(* CODESYS project Avangard(contr5).project
   Title: Avangard(contr1)
   Version: 0.0.0.0
   Author: Administrator

Project tree, tasks and I/O mapping:
  MyController : TM241CE40T/U, Schneider Electric, order no. TM241CE40T/U, version 4.0.6.18
    application Application
      task MAST (cyclic, interval 20 ms, priority 15, watchdog 100 ms x 1) calls MainPrgY, MainLD, MainPrgX
      global variables GVL
    DI : Digital Inputs, Schneider Electric, version 4.0.6.18
        input  idwDI_IDW0 : DWORD  // IDW0
        input  Application.X05_0 : BOOL  // IDW0.I0
        input  Application.X05_1 : BOOL  // IDW0.I1
        input  Application.X05_2 : BOOL  // IDW0.I2
        input  Application.X05_3 : BOOL  // IDW0.I3
        input  Application.X05_4 : BOOL  // IDW0.I4
        input  Application.X05_5 : BOOL  // IDW0.I5
        input  Application.X05_6 : BOOL  // IDW0.I6
        input  Application.X05_7 : BOOL  // IDW0.I7
        input  Application.X05_8 : BOOL  // IDW0.I8
        input  Application.X05_9 : BOOL  // IDW0.I9
        input  Application.X05_10 : BOOL  // IDW0.I10
        input  Application.X05_11 : BOOL  // IDW0.I11
        input  Application.X05_12 : BOOL  // IDW0.I12
        input  Application.X05_13 : BOOL  // IDW0.I13
        input  Application.X05_14 : BOOL  // IDW0.I14
        input  Application.X05_15 : BOOL  // IDW0.I15
        input  Application.X05_16 : BOOL  // IDW0.I16
        input  Application.X05_17 : BOOL  // IDW0.I17
        input  Application.X05_18 : BOOL  // IDW0.I18
        input  Application.X05_19 : BOOL  // IDW0.I19
        input  Application.X05_20 : BOOL  // IDW0.I20
        input  Application.X05_21 : BOOL  // IDW0.I21
        input  Application.X05_22 : BOOL  // IDW0.I22
        input  Application.X05_23 : BOOL  // IDW0.I23
        input  ibDI_IB1 : BYTE  // IB1
    DQ : Digital Outputs, Schneider Electric, version 4.0.6.18
        output Application.Y05_0 : BOOL  // QW0.Q0
        output Application.Y05_1 : BOOL  // QW0.Q1
        output Application.Y05_2 : BOOL  // QW0.Q2
        output Application.Y05_3 : BOOL  // QW0.Q3
        output Application.Y05_4 : BOOL  // QW0.Q4
        output Application.Y05_5 : BOOL  // QW0.Q5
        output Application.Y05_6 : BOOL  // QW0.Q6
        output Application.Y05_7 : BOOL  // QW0.Q7
        output Application.Y05_8 : BOOL  // QW0.Q8
        output Application.Y05_9 : BOOL  // QW0.Q9
        output Application.Y05_10 : BOOL  // QW0.Q10
        output Application.Y05_11 : BOOL  // QW0.Q11
        output Application.Y05_12 : BOOL  // QW0.Q12
        output Application.Y05_13 : BOOL  // QW0.Q13
        output Application.Y05_14 : BOOL  // QW0.Q14
        output Application.Y05_15 : BOOL  // QW0.Q15
        output qbDQ_QB1 : BYTE  // QB1
        unmapped channels: QW0
    Counters : Counters, Schneider Electric, version 4.0.6.18
    Pulse_Generators : Pulse Generators, Schneider Electric, version 4.0.6.18
    Cartridge_1 : Cartridge, Schneider Electric, version 4.0.6.18
    Cartridge_2 : Cartridge, Schneider Electric, version 4.0.6.18
    IO_Bus : IO bus - TM3, Schneider Electric, version 4.0.6.18
      Module_1 : TM3DI32K, Schneider Electric, order no. TM3DI32K, version 1.0.1.3
          input  idwModule_1_ID0 : DWORD  // ID0
          input  Application.X51_0 : BOOL  // ID0.I0
          input  Application.X51_1 : BOOL  // ID0.I1
          input  Application.X51_2 : BOOL  // ID0.I2
          input  Application.X51_3 : BOOL  // ID0.I3
          input  Application.X51_4 : BOOL  // ID0.I4
          input  Application.X51_5 : BOOL  // ID0.I5
          input  Application.X51_6 : BOOL  // ID0.I6
          input  Application.X51_7 : BOOL  // ID0.I7
          input  Application.X51_8 : BOOL  // ID0.I8
          input  Application.X51_9 : BOOL  // ID0.I9
          input  Application.X51_10 : BOOL  // ID0.I10
          input  Application.X51_11 : BOOL  // ID0.I11
          input  Application.X51_12 : BOOL  // ID0.I12
          input  Application.X51_13 : BOOL  // ID0.I13
          input  Application.X51_14 : BOOL  // ID0.I14
          input  Application.X51_15 : BOOL  // ID0.I15
          input  Application.X51_16 : BOOL  // ID0.I16
          input  Application.X51_17 : BOOL  // ID0.I17
          input  Application.X51_18 : BOOL  // ID0.I18
          input  Application.X51_19 : BOOL  // ID0.I19
          input  Application.X51_20 : BOOL  // ID0.I20
          input  Application.X51_21 : BOOL  // ID0.I21
          input  Application.X51_22 : BOOL  // ID0.I22
          input  Application.X51_23 : BOOL  // ID0.I23
          input  Application.X51_24 : BOOL  // ID0.I24
          input  Application.X51_25 : BOOL  // ID0.I25
          input  Application.X51_26 : BOOL  // ID0.I26
          input  Application.X51_27 : BOOL  // ID0.I27
          input  Application.X51_28 : BOOL  // ID0.I28
          input  Application.X51_29 : BOOL  // ID0.I29
          input  Application.X51_30 : BOOL  // ID0.I30
          input  Application.X51_31 : BOOL  // ID0.I31
      Module_2 : TM3DI32K, Schneider Electric, order no. TM3DI32K, version 1.0.1.3
          input  Application.X52_0 : BOOL  // ID0.I0
          input  Application.X52_1 : BOOL  // ID0.I1
          input  Application.X52_2 : BOOL  // ID0.I2
          input  Application.X52_3 : BOOL  // ID0.I3
          input  Application.X52_4 : BOOL  // ID0.I4
          input  Application.X52_5 : BOOL  // ID0.I5
          input  Application.X52_6 : BOOL  // ID0.I6
          input  Application.X52_7 : BOOL  // ID0.I7
          input  Application.X52_8 : BOOL  // ID0.I8
          input  Application.X52_9 : BOOL  // ID0.I9
          input  Application.X52_10 : BOOL  // ID0.I10
          input  Application.X52_11 : BOOL  // ID0.I11
          input  Application.X52_12 : BOOL  // ID0.I12
          input  Application.X52_13 : BOOL  // ID0.I13
          input  Application.X52_14 : BOOL  // ID0.I14
          input  Application.X52_15 : BOOL  // ID0.I15
          input  Application.X52_16 : BOOL  // ID0.I16
          input  Application.X52_17 : BOOL  // ID0.I17
          input  Application.X52_18 : BOOL  // ID0.I18
          input  Application.X52_19 : BOOL  // ID0.I19
          input  Application.X52_20 : BOOL  // ID0.I20
          input  Application.X52_21 : BOOL  // ID0.I21
          input  Application.X52_22 : BOOL  // ID0.I22
          input  Application.X52_23 : BOOL  // ID0.I23
          input  Application.X52_24 : BOOL  // ID0.I24
          input  Application.X52_25 : BOOL  // ID0.I25
          input  Application.X52_26 : BOOL  // ID0.I26
          input  Application.X52_27 : BOOL  // ID0.I27
          input  Application.X52_28 : BOOL  // ID0.I28
          input  Application.X52_29 : BOOL  // ID0.I29
          input  Application.X52_30 : BOOL  // ID0.I30
          input  Application.X52_31 : BOOL  // ID0.I31
          unmapped channels: ID0
      Module_7 : TM3TI4/G, Schneider Electric, order no. TM3TI4/G, version 1.0.1.5
          input  Application.XXa7_0 : INT  // IW0
          input  Application.XXa7_1 : INT  // IW1
          input  Application.XXa7_2 : INT  // IW2
          input  Application.XXa7_3 : INT  // IW3
          input  ibModule_9_IBStatusIW0 : BYTE  // IBStatusIW0
          input  ibModule_9_IBStatusIW1 : BYTE  // IBStatusIW1
          input  ibModule_9_IBStatusIW2 : BYTE  // IBStatusIW2
          input  ibModule_9_IBStatusIW3 : BYTE  // IBStatusIW3
      Module_4 : TM3DI32K, Schneider Electric, order no. TM3DI32K, version 1.0.1.3
          input  Application.X54_0 : BOOL  // ID0.I0
          input  Application.X54_1 : BOOL  // ID0.I1
          input  Application.X54_2 : BOOL  // ID0.I2
          input  Application.X54_3 : BOOL  // ID0.I3
          input  Application.X54_4 : BOOL  // ID0.I4
          input  Application.X54_5 : BOOL  // ID0.I5
          input  Application.X54_6 : BOOL  // ID0.I6
          input  Application.X54_7 : BOOL  // ID0.I7
          input  Application.X54_8 : BOOL  // ID0.I8
          input  Application.X54_9 : BOOL  // ID0.I9
          input  Application.X54_10 : BOOL  // ID0.I10
          input  Application.X54_11 : BOOL  // ID0.I11
          input  Application.X54_12 : BOOL  // ID0.I12
          input  Application.X54_13 : BOOL  // ID0.I13
          input  Application.X54_14 : BOOL  // ID0.I14
          input  Application.X54_15 : BOOL  // ID0.I15
          input  Application.X54_16 : BOOL  // ID0.I16
          input  Application.X54_17 : BOOL  // ID0.I17
          input  Application.X54_18 : BOOL  // ID0.I18
          input  Application.X54_19 : BOOL  // ID0.I19
          input  Application.X54_20 : BOOL  // ID0.I20
          input  Application.X54_21 : BOOL  // ID0.I21
          input  Application.X54_22 : BOOL  // ID0.I22
          input  Application.X54_23 : BOOL  // ID0.I23
          input  Application.X54_24 : BOOL  // ID0.I24
          input  Application.X54_25 : BOOL  // ID0.I25
          input  Application.X54_26 : BOOL  // ID0.I26
          input  Application.X54_27 : BOOL  // ID0.I27
          input  Application.X54_28 : BOOL  // ID0.I28
          input  Application.X54_29 : BOOL  // ID0.I29
          input  Application.X54_30 : BOOL  // ID0.I30
          input  Application.X54_31 : BOOL  // ID0.I31
          unmapped channels: ID0
      Module_3 : TM3DI32K, Schneider Electric, order no. TM3DI32K, version 1.0.1.3
          input  Application.X53_0 : BOOL  // ID0.I0
          input  Application.X53_1 : BOOL  // ID0.I1
          input  Application.X53_2 : BOOL  // ID0.I2
          input  Application.X53_3 : BOOL  // ID0.I3
          input  Application.X53_4 : BOOL  // ID0.I4
          input  Application.X53_5 : BOOL  // ID0.I5
          input  Application.X53_6 : BOOL  // ID0.I6
          input  Application.X53_7 : BOOL  // ID0.I7
          input  Application.X53_8 : BOOL  // ID0.I8
          input  Application.X53_9 : BOOL  // ID0.I9
          input  Application.X53_10 : BOOL  // ID0.I10
          input  Application.X53_11 : BOOL  // ID0.I11
          input  Application.X53_12 : BOOL  // ID0.I12
          input  Application.X53_13 : BOOL  // ID0.I13
          input  Application.X53_14 : BOOL  // ID0.I14
          input  Application.X53_15 : BOOL  // ID0.I15
          input  Application.X53_16 : BOOL  // ID0.I16
          input  Application.X53_17 : BOOL  // ID0.I17
          input  Application.X53_18 : BOOL  // ID0.I18
          input  Application.X53_19 : BOOL  // ID0.I19
          input  Application.X53_20 : BOOL  // ID0.I20
          input  Application.X53_21 : BOOL  // ID0.I21
          input  Application.X53_22 : BOOL  // ID0.I22
          input  Application.X53_23 : BOOL  // ID0.I23
          input  Application.X53_24 : BOOL  // ID0.I24
          input  Application.X53_25 : BOOL  // ID0.I25
          input  Application.X53_26 : BOOL  // ID0.I26
          input  Application.X53_27 : BOOL  // ID0.I27
          input  Application.X53_28 : BOOL  // ID0.I28
          input  Application.X53_29 : BOOL  // ID0.I29
          input  Application.X53_30 : BOOL  // ID0.I30
          input  Application.X53_31 : BOOL  // ID0.I31
          unmapped channels: ID0
      Module_5 : TM3DQ32TK, Schneider Electric, order no. TM3DQ32TK, version 1.0.1.3
          output Application.Y55_0 : BOOL  // QD0.Q0
          output Application.Y55_1 : BOOL  // QD0.Q1
          output Application.Y55_2 : BOOL  // QD0.Q2
          output Application.Y55_3 : BOOL  // QD0.Q3
          output Application.Y55_4 : BOOL  // QD0.Q4
          output Application.Y55_5 : BOOL  // QD0.Q5
          output Application.Y55_6 : BOOL  // QD0.Q6
          output Application.Y55_7 : BOOL  // QD0.Q7
          output Application.Y55_8 : BOOL  // QD0.Q8
          output Application.Y55_9 : BOOL  // QD0.Q9
          output Application.Y55_10 : BOOL  // QD0.Q10
          output Application.Y55_11 : BOOL  // QD0.Q11
          output Application.Y55_12 : BOOL  // QD0.Q12
          output Application.Y55_13 : BOOL  // QD0.Q13
          output Application.Y55_14 : BOOL  // QD0.Q14
          output Application.Y55_15 : BOOL  // QD0.Q15
          output Application.Y55_16 : BOOL  // QD0.Q16
          output Application.Y55_17 : BOOL  // QD0.Q17
          output Application.Y55_18 : BOOL  // QD0.Q18
          output Application.Y55_19 : BOOL  // QD0.Q19
          output Application.Y55_20 : BOOL  // QD0.Q20
          output Application.Y55_21 : BOOL  // QD0.Q21
          output Application.Y55_22 : BOOL  // QD0.Q22
          output Application.Y55_23 : BOOL  // QD0.Q23
          output Application.Y55_24 : BOOL  // QD0.Q24
          output Application.Y55_25 : BOOL  // QD0.Q25
          output Application.Y55_26 : BOOL  // QD0.Q26
          output Application.Y55_27 : BOOL  // QD0.Q27
          output Application.Y55_28 : BOOL  // QD0.Q28
          output Application.Y55_29 : BOOL  // QD0.Q29
          output Application.Y55_30 : BOOL  // QD0.Q30
          output Application.Y55_31 : BOOL  // QD0.Q31
          unmapped channels: QD0
      Module_6 : TM3TI4/G, Schneider Electric, order no. TM3TI4/G, version 1.0.1.5
          input  Application.XXa6_0 : INT  // IW0
          input  Application.XXa6_1 : INT  // IW1
          input  Application.XXa6_2 : INT  // IW2
          input  Application.XXa6_3 : INT  // IW3
          input  ibModule_8_IBStatusIW0 : BYTE  // IBStatusIW0
          input  ibModule_8_IBStatusIW1 : BYTE  // IBStatusIW1
          input  ibModule_8_IBStatusIW2 : BYTE  // IBStatusIW2
          input  ibModule_8_IBStatusIW3 : BYTE  // IBStatusIW3
    COM_Bus : COM bus, Schneider Electric, version 4.0.6.18
    Ethernet_1 : Ethernet Network, Schneider Electric, version 4.0.6.18
        settings: IPAddress = [192, 168, 1, 205]; SubnetMask = [255, 255, 255, 0]; GatewayAddress = [192, 168, 1, 1]; DeviceName = 'TM241CE40T_5'; WebServer = FALSE; FTP Server = FALSE; SoMachine Protocol = TRUE; Modbus Server = TRUE; NetManage Protocol = TRUE; SNMP protocol = FALSE; Enable Routing = FALSE; WebVisu protocol = FALSE; DHCP Server Active = FALSE
    Serial_Line_1 : Serial line, Schneider Electric, version 4.0.6.18
      SoMachine_Network_Manager : SoMachine-Network Manager, Schneider Electric, version 4.0.0.2
    Serial_Line_2 : Serial line, Schneider Electric, version 4.0.6.18
      Modbus_Manager : Modbus Manager, Schneider Electric, version 4.0.0.2
  libraries: Standard, * (System)
  program MainPrgY [ST]
  program MainLD [LD]
  function block DKS [LD]
  program MainPrgX [ST]
*)

// MyController/Application/GVL
VAR_GLOBAL
	XX AT %MW0 : ARRAY[0..9] OF WORD;  //данные с 5го контроллера
	XXa AT %MW10 : ARRAY[0..8] OF INT;  //данные с 5го контроллера
	YY AT %MW18 : ARRAY[0..3] OF WORD;  //данные для 5го контроллера на управление

	DKS_Time : WORD := 3;	//время срабатывания ДКС в сек
	
	Nor10200_DKS : BOOL;
	Nor10400_DKS : BOOL;
	Tr10500_DKS : BOOL;
	Tr10600_DKS : BOOL;
	Tr10700_DKS : BOOL;
	Tr20110_DKS : BOOL;
	Nor20300_DKS : BOOL;
	Nor21200_DKS : BOOL;
	Tr21300_DKS : BOOL;
	Tr30400_DKS : BOOL;
	Nor30500_DKS : BOOL;
	Tr30340_DKS : BOOL;
	Tr30700_DKS : BOOL;
	Nor40100_DKS : BOOL;
	
	
	// Контроллер 1
		//Входа
			X05_0 : BOOL;
			X05_1 : BOOL;
			X05_2 : BOOL;
			X05_3 : BOOL;
			X05_4 : BOOL;
			X05_5 : BOOL;
			X05_6 : BOOL;
			X05_7 : BOOL;
			X05_8 : BOOL;
			X05_9 : BOOL;
			X05_10 : BOOL;
			X05_11 : BOOL;
			X05_12 : BOOL;
			X05_13 : BOOL;
			X05_14 : BOOL;
			X05_15 : BOOL;
			X05_16 : BOOL;
			X05_17 : BOOL;
			X05_18 : BOOL;
			X05_19 : BOOL;
			X05_20 : BOOL;
			X05_21 : BOOL;
			X05_22 : BOOL;
			X05_23 : BOOL;
			X05_24 : BOOL;
			X05_25 : BOOL;
			X05_26 : BOOL;
			X05_27 : BOOL;
			X05_28 : BOOL;
			X05_29 : BOOL;
			X05_30 : BOOL;
			X05_31 : BOOL;
		//Выхода
			Y05_0 : BOOL;
			Y05_1 : BOOL;
			Y05_2 : BOOL;
			Y05_3 : BOOL;
			Y05_4 : BOOL;
			Y05_5 : BOOL;
			Y05_6 : BOOL;
			Y05_7 : BOOL;
			Y05_8 : BOOL;
			Y05_9 : BOOL;
			Y05_10 : BOOL;
			Y05_11 : BOOL;
			Y05_12 : BOOL;
			Y05_13 : BOOL;
			Y05_14 : BOOL;
			Y05_15 : BOOL;
			Y05_16 : BOOL;
			Y05_17 : BOOL;
			Y05_18 : BOOL;
			Y05_19 : BOOL;
			Y05_20 : BOOL;
			Y05_21 : BOOL;
			Y05_22 : BOOL;
			Y05_23 : BOOL;
			Y05_24 : BOOL;
			Y05_25 : BOOL;
			Y05_26 : BOOL;
			Y05_27 : BOOL;
			Y05_28 : BOOL;
			Y05_29 : BOOL;
			Y05_30 : BOOL;
			Y05_31 : BOOL;
			
	// Модуль расширения 1 контроллер 1 
		//Входа
			X51_0 : BOOL;
			X51_1 : BOOL;
			X51_2 : BOOL;
			X51_3 : BOOL;
			X51_4 : BOOL;
			X51_5 : BOOL;
			X51_6 : BOOL;
			X51_7 : BOOL;
			X51_8 : BOOL;
			X51_9 : BOOL;
			X51_10 : BOOL;
			X51_11 : BOOL;
			X51_12 : BOOL;
			X51_13 : BOOL;
			X51_14 : BOOL;
			X51_15 : BOOL;
			X51_16 : BOOL;
			X51_17 : BOOL;
			X51_18 : BOOL;
			X51_19 : BOOL;
			X51_20 : BOOL;
			X51_21 : BOOL;
			X51_22 : BOOL;
			X51_23 : BOOL;
			X51_24 : BOOL;
			X51_25 : BOOL;
			X51_26 : BOOL;
			X51_27 : BOOL;
			X51_28 : BOOL;
			X51_29 : BOOL;
			X51_30 : BOOL;
			X51_31 : BOOL;
		//Выхода
			Y51_0 : BOOL;
			Y51_1 : BOOL;
			Y51_2 : BOOL;
			Y51_3 : BOOL;
			Y51_4 : BOOL;
			Y51_5 : BOOL;
			Y51_6 : BOOL;
			Y51_7 : BOOL;
			Y51_8 : BOOL;
			Y51_9 : BOOL;
			Y51_10 : BOOL;
			Y51_11 : BOOL;
			Y51_12 : BOOL;
			Y51_13 : BOOL;
			Y51_14 : BOOL;
			Y51_15 : BOOL;
			Y51_16 : BOOL;
			Y51_17 : BOOL;
			Y51_18 : BOOL;
			Y51_19 : BOOL;
			Y51_20 : BOOL;
			Y51_21 : BOOL;
			Y51_22 : BOOL;
			Y51_23 : BOOL;
			Y51_24 : BOOL;
			Y51_25 : BOOL;
			Y51_26 : BOOL;
			Y51_27 : BOOL;
			Y51_28 : BOOL;
			Y51_29 : BOOL;
			Y51_30 : BOOL;
			Y51_31 : BOOL;
	
	// Модуль расширения 2 контроллер 1
		//Входа
			X52_0 : BOOL;
			X52_1 : BOOL;
			X52_2 : BOOL;
			X52_3 : BOOL;
			X52_4 : BOOL;
			X52_5 : BOOL;
			X52_6 : BOOL;
			X52_7 : BOOL;
			X52_8 : BOOL;
			X52_9 : BOOL;
			X52_10 : BOOL;
			X52_11 : BOOL;
			X52_12 : BOOL;
			X52_13 : BOOL;
			X52_14 : BOOL;
			X52_15 : BOOL;
			X52_16 : BOOL;
			X52_17 : BOOL;
			X52_18 : BOOL;
			X52_19 : BOOL;
			X52_20 : BOOL;
			X52_21 : BOOL;
			X52_22 : BOOL;
			X52_23 : BOOL;
			X52_24 : BOOL;
			X52_25 : BOOL;
			X52_26 : BOOL;
			X52_27 : BOOL;
			X52_28 : BOOL;
			X52_29 : BOOL;
			X52_30 : BOOL;
			X52_31 : BOOL;
		//Выхода
			Y52_0 : BOOL;
			Y52_1 : BOOL;
			Y52_2 : BOOL;
			Y52_3 : BOOL;
			Y52_4 : BOOL;
			Y52_5 : BOOL;
			Y52_6 : BOOL;
			Y52_7 : BOOL;
			Y52_8 : BOOL;
			Y52_9 : BOOL;
			Y52_10 : BOOL;
			Y52_11 : BOOL;
			Y52_12 : BOOL;
			Y52_13 : BOOL;
			Y52_14 : BOOL;
			Y52_15 : BOOL;
			Y52_16 : BOOL;
			Y52_17 : BOOL;
			Y52_18 : BOOL;
			Y52_19 : BOOL;
			Y52_20 : BOOL;
			Y52_21 : BOOL;
			Y52_22 : BOOL;
			Y52_23 : BOOL;
			Y52_24 : BOOL;
			Y52_25 : BOOL;
			Y52_26 : BOOL;
			Y52_27 : BOOL;
			Y52_28 : BOOL;
			Y52_29 : BOOL;
			Y52_30 : BOOL;
			Y52_31 : BOOL;
			
	// Модуль расширения 3 контроллер 1
		//Входа
			X53_0 : BOOL;
			X53_1 : BOOL;
			X53_2 : BOOL;
			X53_3 : BOOL;
			X53_4 : BOOL;
			X53_5 : BOOL;
			X53_6 : BOOL;
			X53_7 : BOOL;
			X53_8 : BOOL;
			X53_9 : BOOL;
			X53_10 : BOOL;
			X53_11 : BOOL;
			X53_12 : BOOL;
			X53_13 : BOOL;
			X53_14 : BOOL;
			X53_15 : BOOL;
			X53_16 : BOOL;
			X53_17 : BOOL;
			X53_18 : BOOL;
			X53_19 : BOOL;
			X53_20 : BOOL;
			X53_21 : BOOL;
			X53_22 : BOOL;
			X53_23 : BOOL;
			X53_24 : BOOL;
			X53_25 : BOOL;
			X53_26 : BOOL;
			X53_27 : BOOL;
			X53_28 : BOOL;
			X53_29 : BOOL;
			X53_30 : BOOL;
			X53_31 : BOOL;
		//Выхода
			Y53_0 : BOOL;
			Y53_1 : BOOL;
			Y53_2 : BOOL;
			Y53_3 : BOOL;
			Y53_4 : BOOL;
			Y53_5 : BOOL;
			Y53_6 : BOOL;
			Y53_7 : BOOL;
			Y53_8 : BOOL;
			Y53_9 : BOOL;
			Y53_10 : BOOL;
			Y53_11 : BOOL;
			Y53_12 : BOOL;
			Y53_13 : BOOL;
			Y53_14 : BOOL;
			Y53_15 : BOOL;
			Y53_16 : BOOL;
			Y53_17 : BOOL;
			Y53_18 : BOOL;
			Y53_19 : BOOL;
			Y53_20 : BOOL;
			Y53_21 : BOOL;
			Y53_22 : BOOL;
			Y53_23 : BOOL;
			Y53_24 : BOOL;
			Y53_25 : BOOL;
			Y53_26 : BOOL;
			Y53_27 : BOOL;
			Y53_28 : BOOL;
			Y53_29 : BOOL;
			Y53_30 : BOOL;
			Y53_31 : BOOL;			

	// Модуль расширения 4 контроллер 1
		//Входа
			X54_0 : BOOL;
			X54_1 : BOOL;
			X54_2 : BOOL;
			X54_3 : BOOL;
			X54_4 : BOOL;
			X54_5 : BOOL;
			X54_6 : BOOL;
			X54_7 : BOOL;
			X54_8 : BOOL;
			X54_9 : BOOL;
			X54_10 : BOOL;
			X54_11 : BOOL;
			X54_12 : BOOL;
			X54_13 : BOOL;
			X54_14 : BOOL;
			X54_15 : BOOL;
			X54_16 : BOOL;
			X54_17 : BOOL;
			X54_18 : BOOL;
			X54_19 : BOOL;
			X54_20 : BOOL;
			X54_21 : BOOL;
			X54_22 : BOOL;
			X54_23 : BOOL;
			X54_24 : BOOL;
			X54_25 : BOOL;
			X54_26 : BOOL;
			X54_27 : BOOL;
			X54_28 : BOOL;
			X54_29 : BOOL;
			X54_30 : BOOL;
			X54_31 : BOOL;
		//Выхода
			Y54_0 : BOOL;
			Y54_1 : BOOL;
			Y54_2 : BOOL;
			Y54_3 : BOOL;
			Y54_4 : BOOL;
			Y54_5 : BOOL;
			Y54_6 : BOOL;
			Y54_7 : BOOL;
			Y54_8 : BOOL;
			Y54_9 : BOOL;
			Y54_10 : BOOL;
			Y54_11 : BOOL;
			Y54_12 : BOOL;
			Y54_13 : BOOL;
			Y54_14 : BOOL;
			Y54_15 : BOOL;
			Y54_16 : BOOL;
			Y54_17 : BOOL;
			Y54_18 : BOOL;
			Y54_19 : BOOL;
			Y54_20 : BOOL;
			Y54_21 : BOOL;
			Y54_22 : BOOL;
			Y54_23 : BOOL;
			Y54_24 : BOOL;
			Y54_25 : BOOL;
			Y54_26 : BOOL;
			Y54_27 : BOOL;
			Y54_28 : BOOL;
			Y54_29 : BOOL;
			Y54_30 : BOOL;
			Y54_31 : BOOL;
	// Модуль расширения 5 контроллер 1
		//Входа
			X55_0 : BOOL;
			X55_1 : BOOL;
			X55_2 : BOOL;
			X55_3 : BOOL;
			X55_4 : BOOL;
			X55_5 : BOOL;
			X55_6 : BOOL;
			X55_7 : BOOL;
			X55_8 : BOOL;
			X55_9 : BOOL;
			X55_10 : BOOL;
			X55_11 : BOOL;
			X55_12 : BOOL;
			X55_13 : BOOL;
			X55_14 : BOOL;
			X55_15 : BOOL;
			X55_16 : BOOL;
			X55_17 : BOOL;
			X55_18 : BOOL;
			X55_19 : BOOL;
			X55_20 : BOOL;
			X55_21 : BOOL;
			X55_22 : BOOL;
			X55_23 : BOOL;
			X55_24 : BOOL;
			X55_25 : BOOL;
			X55_26 : BOOL;
			X55_27 : BOOL;
			X55_28 : BOOL;
			X55_29 : BOOL;
			X55_30 : BOOL;
			X55_31 : BOOL;
		//Выхода
			Y55_0 : BOOL;
			Y55_1 : BOOL;
			Y55_2 : BOOL;
			Y55_3 : BOOL;
			Y55_4 : BOOL;
			Y55_5 : BOOL;
			Y55_6 : BOOL;
			Y55_7 : BOOL;
			Y55_8 : BOOL;
			Y55_9 : BOOL;
			Y55_10 : BOOL;
			Y55_11 : BOOL;
			Y55_12 : BOOL;
			Y55_13 : BOOL;
			Y55_14 : BOOL;
			Y55_15 : BOOL;
			Y55_16 : BOOL;
			Y55_17 : BOOL;
			Y55_18 : BOOL;
			Y55_19 : BOOL;
			Y55_20 : BOOL;
			Y55_21 : BOOL;
			Y55_22 : BOOL;
			Y55_23 : BOOL;
			Y55_24 : BOOL;
			Y55_25 : BOOL;
			Y55_26 : BOOL;
			Y55_27 : BOOL;
			Y55_28 : BOOL;
			Y55_29 : BOOL;
			Y55_30 : BOOL;
			Y55_31 : BOOL;
	// Модуль расширения 6 контроллер 1
		//Входа
			X56_0 : BOOL;
			X56_1 : BOOL;
			X56_2 : BOOL;
			X56_3 : BOOL;
			X56_4 : BOOL;
			X56_5 : BOOL;
			X56_6 : BOOL;
			X56_7 : BOOL;
			X56_8 : BOOL;
			X56_9 : BOOL;
			X56_10 : BOOL;
			X56_11 : BOOL;
			X56_12 : BOOL;
			X56_13 : BOOL;
			X56_14 : BOOL;
			X56_15 : BOOL;
			X56_16 : BOOL;
			X56_17 : BOOL;
			X56_18 : BOOL;
			X56_19 : BOOL;
			X56_20 : BOOL;
			X56_21 : BOOL;
			X56_22 : BOOL;
			X56_23 : BOOL;
			X56_24 : BOOL;
			X56_25 : BOOL;
			X56_26 : BOOL;
			X56_27 : BOOL;
			X56_28 : BOOL;
			X56_29 : BOOL;
			X56_30 : BOOL;
			X56_31 : BOOL;
		//Выхода
			Y56_0 : BOOL;
			Y56_1 : BOOL;
			Y56_2 : BOOL;
			Y56_3 : BOOL;
			Y56_4 : BOOL;
			Y56_5 : BOOL;
			Y56_6 : BOOL;
			Y56_7 : BOOL;
			Y56_8 : BOOL;
			Y56_9 : BOOL;
			Y56_10 : BOOL;
			Y56_11 : BOOL;
			Y56_12 : BOOL;
			Y56_13 : BOOL;
			Y56_14 : BOOL;
			Y56_15 : BOOL;
			Y56_16 : BOOL;
			Y56_17 : BOOL;
			Y56_18 : BOOL;
			Y56_19 : BOOL;
			Y56_20 : BOOL;
			Y56_21 : BOOL;
			Y56_22 : BOOL;
			Y56_23 : BOOL;
			Y56_24 : BOOL;
			Y56_25 : BOOL;
			Y56_26 : BOOL;
			Y56_27 : BOOL;
			Y56_28 : BOOL;
			Y56_29 : BOOL;
			Y56_30 : BOOL;
			Y56_31 : BOOL;

	// Модуль расширения 7 контроллер 1
		//Входа
			X57_0 : BOOL;
			X57_1 : BOOL;
			X57_2 : BOOL;
			X57_3 : BOOL;
			X57_4 : BOOL;
			X57_5 : BOOL;
			X57_6 : BOOL;
			X57_7 : BOOL;
			X57_8 : BOOL;
			X57_9 : BOOL;
			X57_10 : BOOL;
			X57_11 : BOOL;
			X57_12 : BOOL;
			X57_13 : BOOL;
			X57_14 : BOOL;
			X57_15 : BOOL;
			X57_16 : BOOL;
			X57_17 : BOOL;
			X57_18 : BOOL;
			X57_19 : BOOL;
			X57_20 : BOOL;
			X57_21 : BOOL;
			X57_22 : BOOL;
			X57_23 : BOOL;
			X57_24 : BOOL;
			X57_25 : BOOL;
			X57_26 : BOOL;
			X57_27 : BOOL;
			X57_28 : BOOL;
			X57_29 : BOOL;
			X57_30 : BOOL;
			X57_31 : BOOL;
		//Выхода
			Y57_0 : BOOL;
			Y57_1 : BOOL;
			Y57_2 : BOOL;
			Y57_3 : BOOL;
			Y57_4 : BOOL;
			Y57_5 : BOOL;
			Y57_6 : BOOL;
			Y57_7 : BOOL;
			Y57_8 : BOOL;
			Y57_9 : BOOL;
			Y57_10 : BOOL;
			Y57_11 : BOOL;
			Y57_12 : BOOL;
			Y57_13 : BOOL;
			Y57_14 : BOOL;
			Y57_15 : BOOL;
			Y57_16 : BOOL;
			Y57_17 : BOOL;
			Y57_18 : BOOL;
			Y57_19 : BOOL;
			Y57_20 : BOOL;
			Y57_21 : BOOL;
			Y57_22 : BOOL;
			Y57_23 : BOOL;
			Y57_24 : BOOL;
			Y57_25 : BOOL;
			Y57_26 : BOOL;
			Y57_27 : BOOL;
			Y57_28 : BOOL;
			Y57_29 : BOOL;
			Y57_30 : BOOL;
			Y57_31 : BOOL;
			
	XXa6_0 : INT;
	XXa6_1 : INT;
	XXa6_2 : INT;
	XXa6_3 : INT;
	XXa7_0 : INT;
	XXa7_1 : INT;
	XXa7_2 : INT;
	XXa7_3 : INT;

END_VAR

// MainPrgY
PROGRAM MainPrgY
VAR
END_VAR

	//выходы
		Y05_0 := YY[0].0;		
		Y05_1 := YY[0].1;
		Y05_2 := YY[0].2;
		Y05_3 := YY[0].3;
		Y05_4 := YY[0].4;
		Y05_5 := YY[0].5;
		Y05_6 := YY[0].6;
		Y05_7 := YY[0].7;
		Y05_8 := YY[0].8;
		Y05_9 := YY[0].9;
		Y05_10 := YY[0].10;
		Y05_11 := YY[0].11;
		Y05_12 := YY[0].12;
		Y05_13 := YY[0].13;
		Y05_14 := YY[0].14;
		Y05_15 := YY[0].15;
		Y05_16 := YY[1].0;
		Y05_17 := YY[1].1;
		Y05_18 := YY[1].2;
		Y05_19 := YY[1].3;
		Y05_20 := YY[1].4;
		Y05_21 := YY[1].5;
		Y05_22 := YY[1].6;
		Y05_23 := YY[1].7;
		Y05_24 := YY[1].8;
		Y05_25 := YY[1].9;
		Y05_26 := YY[1].10;
		Y05_27 := YY[1].11;
		Y05_28 := YY[1].12;
		Y05_29 := YY[1].13;
		Y05_30 := YY[1].14;
		Y05_31 := YY[1].15;
		
		Y55_0 := YY[2].0;		
		Y55_1 := YY[2].1;
		Y55_2 := YY[2].2;
		Y55_3 := YY[2].3;
		Y55_4 := YY[2].4;
		Y55_5 := YY[2].5;
		Y55_6 := YY[2].6;
		Y55_7 := YY[2].7;
		Y55_8 := YY[2].8;
		Y55_9 := YY[2].9;
		Y55_10 := YY[2].10;
		Y55_11 := YY[2].11;
		Y55_12 := YY[2].12;
		Y55_13 := YY[2].13;
		Y55_14 := YY[2].14;
		Y55_15 := YY[2].15;
		Y55_16 := YY[3].0;
		Y55_17 := YY[3].1;
		Y55_18 := YY[3].2;
		Y55_19 := YY[3].3;
		Y55_20 := YY[3].4;
		Y55_21 := YY[3].5;
		Y55_22 := YY[3].6;
		Y55_23 := YY[3].7;
		Y55_24 := YY[3].8;
		Y55_25 := YY[3].9;
		Y55_26 := YY[3].10;
		Y55_27 := YY[3].11;
		Y55_28 := YY[3].12;
		Y55_29 := YY[3].13;
		Y55_30 := YY[3].14;
		Y55_31 := YY[3].15;

END_PROGRAM

// MainLD
PROGRAM MainLD
VAR
	DKS_Nor10200: DKS;
	DKS_Nor10400: DKS;
	DKS_Tr10500: DKS;
	DKS_Tr10600: DKS;
	DKS_Tr10700: DKS;
	DKS_Tr20110: DKS;
	DKS_Nor20300: DKS;
	DKS_Nor21200: DKS;
	DKS_Tr21300: DKS;
	DKS_Tr30400: DKS;
	DKS_Nor30500: DKS;
	DKS_Tr30340: DKS;
	DKS_Tr30700: DKS;
	DKS_Nor40100: DKS;
END_VAR

// NETWORK 1

// NETWORK 2

// NETWORK 3

// NETWORK 4

// NETWORK 5

// NETWORK 6

END_PROGRAM

// DKS
FUNCTION_BLOCK DKS
VAR_INPUT
	Run : BOOL;
	xDks : BOOL;
	TimeDks : WORD;
END_VAR

VAR_OUTPUT
	ErrDks : BOOL;
END_VAR
VAR
	TON_DKS_ON: TON;
	TON_DKS_OFF: TON;
END_VAR

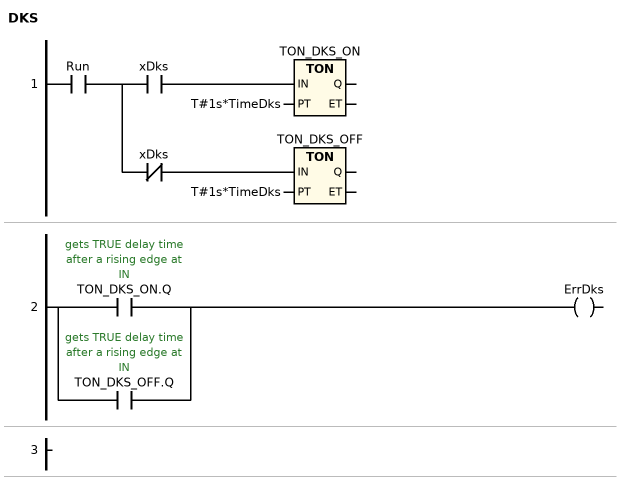
// NETWORK 1
TON_DKS_ON(IN := Run AND xDks, PT := T#1s*TimeDks); // TON
TON_DKS_OFF(IN := Run AND NOT xDks, PT := T#1s*TimeDks); // TON

// NETWORK 2
//   TON_DKS_ON.Q: gets TRUE delay time after a rising edge at IN
//   TON_DKS_OFF.Q: gets TRUE delay time after a rising edge at IN
ErrDks := TON_DKS_ON.Q OR TON_DKS_OFF.Q;

// NETWORK 3

END_FUNCTION_BLOCK

// MainPrgX
PROGRAM MainPrgX
VAR
END_VAR

		XX[0].0 := X05_0;
		XX[0].1 := X05_1;
		XX[0].2 := X05_2;
		XX[0].3 := X05_3;
		XX[0].4 := X05_4;
		XX[0].5 := X05_5;
		XX[0].6 := X05_6;
		XX[0].7 := X05_7;
		XX[0].8 := X05_8;
		XX[0].9 := X05_9;
		XX[0].10 := X05_10;
		XX[0].11 := X05_11;
		XX[0].12 := X05_12;
		XX[0].13 := X05_13;
		XX[0].14 := X05_14;
		XX[0].15 := X05_15;
		XX[1].0 := X05_16;
		XX[1].1 := X05_17;
		XX[1].2 := X05_18;
		XX[1].3 := X05_19;
		XX[1].4 := X05_20;
		XX[1].5 := X05_21;
		XX[1].6 := X05_22;
		XX[1].7 := X05_23;
		XX[1].8 := X05_24;
		XX[1].9 := X05_25;
		XX[1].10 := X05_26;
		XX[1].11 := X05_27;
		XX[1].12 := X05_28;
		XX[1].13 := X05_29;
		XX[1].14 := X05_30;
		XX[1].15 := X05_31;
		
		XX[2].0 := X51_0;
		XX[2].1 := X51_1;
		XX[2].2 := X51_2;
		XX[2].3 := X51_3;
		XX[2].4 := X51_4;
		XX[2].5 := X51_5;
		XX[2].6 := X51_6;
		XX[2].7 := X51_7;
		XX[2].8 := X51_8;
		XX[2].9 := X51_9;
		XX[2].10 := X51_10;
		XX[2].11 := X51_11;
		XX[2].12 := X51_12;
		XX[2].13 := X51_13;
		XX[2].14 := X51_14;
		XX[2].15 := X51_15;
		XX[3].0 := X51_16;
		XX[3].1 := X51_17;
		XX[3].2 := X51_18;
		XX[3].3 := X51_19;
		XX[3].4 := X51_20;
		XX[3].5 := X51_21;
		XX[3].6 := X51_22;
		XX[3].7 := X51_23;
		XX[3].8 := X51_24;
		XX[3].9 := X51_25;
		XX[3].10 := X51_26;
		XX[3].11 := X51_27;
		XX[3].12 := X51_28;
		XX[3].13 := X51_29;
		XX[3].14 := X51_30;
		XX[3].15 := X51_31;
		
		XX[4].0 := X52_0;
		XX[4].1 := X52_1;
		XX[4].2 := X52_2;
		XX[4].3 := X52_3;
		XX[4].4 := X52_4;
		XX[4].5 := X52_5;
		XX[4].6 := X52_6;
		XX[4].7 := X52_7;
		XX[4].8 := X52_8;
		XX[4].9 := X52_9;
		XX[4].10 := X52_10;
		XX[4].11 := X52_11;
		XX[4].12 := X52_12;
		XX[4].13 := X52_13;
		XX[4].14 := X52_14;
		XX[4].15 := X52_15;
		XX[5].0 := X52_16;
		XX[5].1 := X52_17;
		XX[5].2 := X52_18;
		XX[5].3 := X52_19;
		XX[5].4 := X52_20;
		XX[5].5 := X52_21;
		XX[5].6 := X52_22;
		XX[5].7 := X52_23;
		XX[5].8 := X52_24;
		XX[5].9 := X52_25;
		XX[5].10 := X52_26;
		XX[5].11 := X52_27;
		XX[5].12 := X52_28;
		XX[5].13 := X52_29;
		XX[5].14 := X52_30;
		XX[5].15 := X52_31;
		
		XX[6].0 := X53_0;
		XX[6].1 := X53_1;
		XX[6].2 := X53_2;
		XX[6].3 := X53_3;
		XX[6].4 := X53_4;
		XX[6].5 := X53_5;
		XX[6].6 := X53_6;
		XX[6].7 := X53_7;
		XX[6].8 := X53_8;
		XX[6].9 := X53_9;
		XX[6].10 := X53_10;
		XX[6].11 := X53_11;
		XX[6].12 := X53_12;
		XX[6].13 := X53_13;
		XX[6].14 := X53_14;
		XX[6].15 := X53_15;
		XX[7].0 := X53_16;
		XX[7].1 := X53_17;
		XX[7].2 := X53_18;
		XX[7].3 := X53_19;
		XX[7].4 := X53_20;
		XX[7].5 := X53_21;
		XX[7].6 := X53_22;
		XX[7].7 := X53_23;
		XX[7].8 := X53_24;
		XX[7].9 := X53_25;
		XX[7].10 := X53_26;
		XX[7].11 := X53_27;
		XX[7].12 := X53_28;
		XX[7].13 := X53_29;
		XX[7].14 := X53_30;
		XX[7].15 := X53_31;
		
		XX[8].0 := X54_0;
		XX[8].1 := X54_1;
		XX[8].2 := X54_2;
		XX[8].3 := X54_3;
		XX[8].4 := X54_4;
		XX[8].5 := X54_5;
		XX[8].6 := X54_6;
		XX[8].7 := X54_7;
		XX[8].8 := X54_8;
		XX[8].9 := X54_9;
		XX[8].10 := X54_10;
		XX[8].11 := X54_11;
		XX[8].12 := X54_12;
		XX[8].13 := X54_13;
		XX[8].14 := X54_14;
		XX[8].15 := X54_15;
		XX[9].0 := X54_16;
		XX[9].1 := X54_17;
		XX[9].2 := X54_18;
		XX[9].3 := X54_19;
		XX[9].4 := X54_20;
		XX[9].5 := X54_21;
		XX[9].6 := X54_22;
		XX[9].7 := X54_23;
		XX[9].8 := X54_24;
		XX[9].9 := X54_25;
		XX[9].10 := X54_26;
		XX[9].11 := X54_27;
		XX[9].12 := X54_28;
		XX[9].13 := X54_29;
		XX[9].14 := X54_30;
		XX[9].15 := X54_31;
		
		XXa[0]:=XXa6_0;
		XXa[1]:=XXa6_1;
		XXa[2]:=XXa6_2;
		XXa[3]:=XXa6_3;
		XXa[4]:=XXa7_0;
		XXa[5]:=XXa7_1;
		XXa[6]:=XXa7_2;
		XXa[7]:=XXa7_3;

END_PROGRAM
